FUNCTION_BLOCK RemoteTriggeredClock (* Used to initialize/update a time stamp and start a clock remotely. *)
  (* Standard: 61499-2 *)
  (* Version 1.0, 2017-08-27, Marc Jakobi, HTW Berlin *)
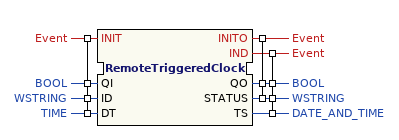
  EVENT_INPUT
    INIT WITH QI, ID, DT; (* Initialization Request *)
  END_EVENT
  EVENT_OUTPUT
    INITO WITH QO, STATUS; (* Initialization Confirm *)
    IND WITH QO, TS, STATUS; (* Execution Confirmation *)
  END_EVENT
  VAR_INPUT
    QI : BOOL; (* Input event qualifier *)
    ID : WSTRING; (* Connection identifier *)
    DT : TIME; (* Tick rate *)
  END_VAR
  VAR_OUTPUT
    QO : BOOL; (* Output event qualifier *)
    STATUS : WSTRING; (* Service status *)
    TS : DATE_AND_TIME; (* Time stamp *)
  END_VAR
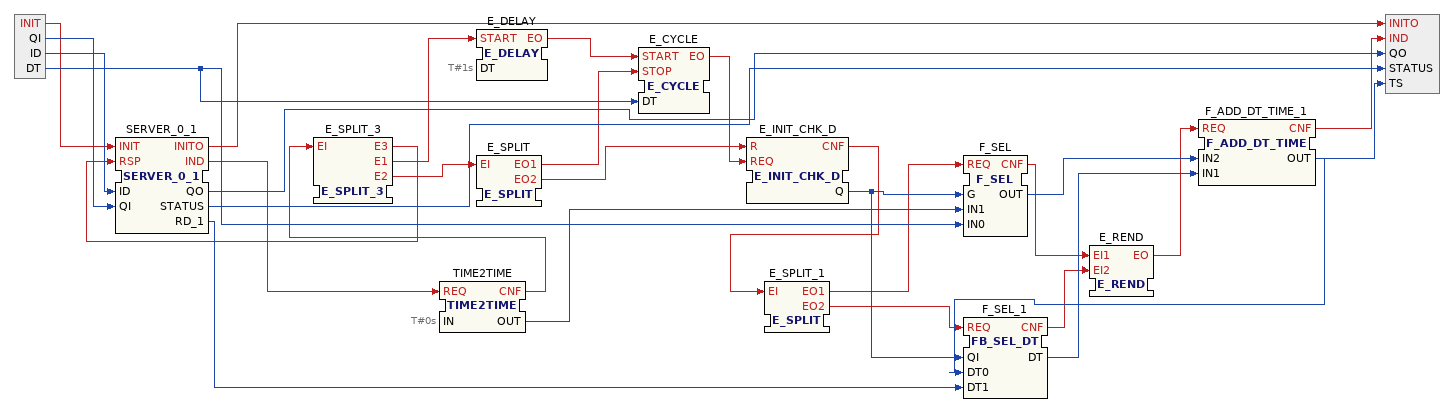
  FBS
    SERVER_0_1 : SERVER_0_1;
    E_SPLIT_3 : E_SPLIT_3;
    TIME2TIME : TIME2TIME(IN := T#0s);
    E_DELAY : E_DELAY(DT := T#1s);
    E_CYCLE : E_CYCLE;
    E_SPLIT : E_SPLIT;
    E_INIT_CHK_D : E_INIT_CHK_D;
    E_SPLIT_1 : E_SPLIT;
    F_SEL : F_SEL;
    E_REND : E_REND;
    F_ADD_DT_TIME_1 : F_ADD_DT_TIME;
    F_SEL_1 : FB_SEL_DT;
  END_FBS
  EVENT_CONNECTIONS
    INIT TO SERVER_0_1.INIT;
    TIME2TIME.CNF TO E_SPLIT_3.EI;
    E_SPLIT_3.E3 TO SERVER_0_1.RSP;
    E_SPLIT_3.E1 TO E_DELAY.START;
    E_DELAY.EO TO E_CYCLE.START;
    E_SPLIT_3.E2 TO E_SPLIT.EI;
    E_SPLIT.EO1 TO E_CYCLE.STOP;
    E_SPLIT.EO2 TO E_INIT_CHK_D.R;
    E_CYCLE.EO TO E_INIT_CHK_D.REQ;
    E_INIT_CHK_D.CNF TO E_SPLIT_1.EI;
    E_SPLIT_1.EO1 TO F_SEL.REQ;
    F_SEL.CNF TO E_REND.EI1;
    E_REND.EO TO F_ADD_DT_TIME_1.REQ;
    F_ADD_DT_TIME_1.CNF TO IND;
    SERVER_0_1.INITO TO INITO;
    E_SPLIT_1.EO2 TO F_SEL_1.REQ;
    F_SEL_1.CNF TO E_REND.EI2;
    SERVER_0_1.IND TO TIME2TIME.REQ;
  END_CONNECTIONS
  DATA_CONNECTIONS
    ID TO SERVER_0_1.ID;
    QI TO SERVER_0_1.QI;
    DT TO E_CYCLE.DT;
    E_INIT_CHK_D.Q TO F_SEL.G;
    TIME2TIME.OUT TO F_SEL.IN1;
    DT TO F_SEL.IN0;
    F_ADD_DT_TIME_1.OUT TO TS;
    SERVER_0_1.QO TO QO;
    SERVER_0_1.STATUS TO STATUS;
    F_SEL.OUT TO F_ADD_DT_TIME_1.IN2;
    E_INIT_CHK_D.Q TO F_SEL_1.QI;
    F_ADD_DT_TIME_1.OUT TO F_SEL_1.DT0;
    SERVER_0_1.RD_1 TO F_SEL_1.DT1;
    F_SEL_1.DT TO F_ADD_DT_TIME_1.IN1;
  END_CONNECTIONS
END_FUNCTION_BLOCK
